// TIA Portal V18 export
TYPE "typeTokenRow"
TITLE = typeTokenRow
// use case specific structure for TDS token row
   STRUCT
      Pressure { ExternalAccessible := 'False'; ExternalVisible := 'False'; ExternalWritable := 'False'} : Int;   // row value for column 'Amount'
      Temperature { ExternalAccessible := 'False'; ExternalVisible := 'False'; ExternalWritable := 'False'} : Int;   // row value for column 'Color'
   END_STRUCT;
END_TYPE
